Universal Robots PolyScope program: Short_LidToCamera.urp

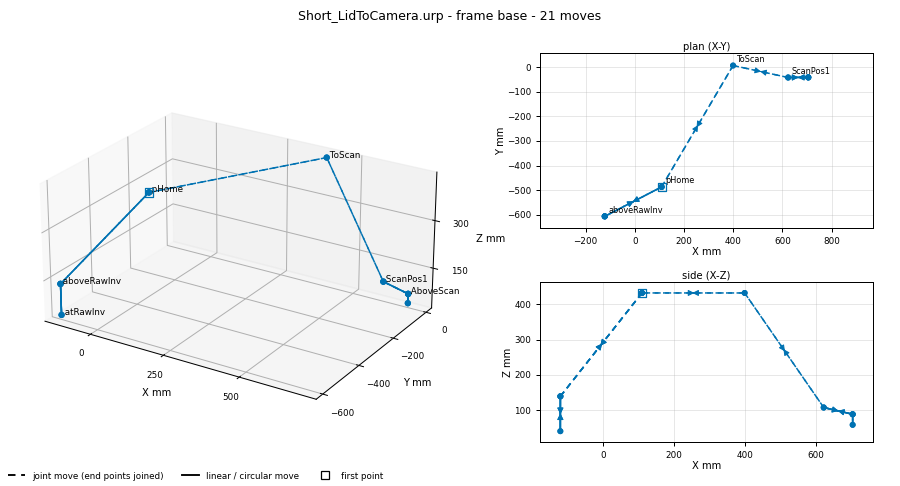
[picture p0: tool path of Short_LidToCamera.urp in frame base, 21 of 21 moves have a stored position in this frame; points joined in program order, loops and branches not executed]
Program Short_LidToCamera (installation=admin directory=/programs/THU_530PM/Final createdIn=3.8.0.61336 lastSavedIn=3.15.8.106339 robotSerialNumber=2015350926)
Calibrated DH parameters: a=[0, -0.425, -0.39225, 0, 0, 0]; d=[0.089159, 0, 0, 0.10915, 0.09465, 0.0823]; alpha=[1.570796, 0, 0, 1.570796, -1.570796, 0]; deltaTheta=[0, 0, 0, 0, 0, 0]
Robot Program (runOnlyOnce=true)
  Set DigitalOutput pin=digital_out[0]; digitalValue=0
  MoveJ speed 180 deg/s, acceleration 200 deg/s^2 (useActiveTCP=true)
    Waypoint pHome: TCP in base x=109.083 y=-486.882 z=431.849 mm, rx=0.0001 ry=3.1416 rz=-0.0001 rad; joints [89.992, -90.005, 90.008, -90.008, -90, -0.005] deg
    Call _adminLinearIndex1
    Waypoint aboveRawInv: TCP in base x=-121.786 y=-606.279 z=139.423 mm, rx=2.2213 ry=2.2177 rz=-0.001 rad; joints [68.458, -61.321, 99.13, -127.905, -89.867, 68.551] deg
  MoveL speed 250 mm/s, acceleration 1200 mm/s^2 (useActiveTCP=true) feature=Base
    Waypoint atRawInv: TCP in base x=-121.937 y=-606.364 z=40.769 mm, rx=2.2227 ry=2.216 rz=-0.0011 rad; joints [68.446, -51.912, 101.978, -140.169, -89.857, 68.619] deg
    Set DigitalOutput pin=digital_out[0]; digitalValue=1
    Wait Sleep waitTime=1
    Waypoint aboveRawInv: TCP in base x=-121.786 y=-606.279 z=139.423 mm, rx=2.2213 ry=2.2177 rz=-0.001 rad; joints [68.458, -61.321, 99.13, -127.905, -89.867, 68.551] deg
  MoveJ speed 180 deg/s, acceleration 200 deg/s^2 (useActiveTCP=true)
    Waypoint pHome: TCP in base x=109.083 y=-486.882 z=431.849 mm, rx=0.0001 ry=3.1416 rz=-0.0001 rad; joints [89.992, -90.005, 90.008, -90.008, -90, -0.005] deg
  Call _adminLinearIndex1
  MoveJ speed 60 deg/s, acceleration 80 deg/s^2 (useActiveTCP=true)
    Waypoint ToScan: TCP in base x=399.431 y=6.288 z=431.784 mm, rx=0 ry=-3.1415 rz=0 rad; joints [165.046, -103.944, 102.123, -88.173, -90.001, 75.046] deg
    Waypoint ScanPos1: TCP in base x=623.056 y=-42.326 z=107.794 mm, rx=0.0456 ry=-3.1308 rz=0.0038 rad; joints [166.086, -57.904, 99.074, -130.624, -90.289, 74.42] deg
  MoveL speed 250 mm/s, acceleration 1200 mm/s^2 (useActiveTCP=true) feature=Base
    Waypoint AboveScan: TCP in base x=704.91 y=-41.789 z=88.68 mm, rx=0.0458 ry=-3.1307 rz=0.0039 rad; joints [167.748, -47.56, 83.623, -125.504, -90.275, 76.074] deg
    Waypoint AtScan: TCP in base x=704.921 y=-41.77 z=58.801 mm, rx=0.0456 ry=-3.1306 rz=0.0038 rad; joints [167.749, -45.085, 84.321, -128.675, -90.272, 76.08] deg
    Set DigitalOutput pin=digital_out[0]; digitalValue=0
    Wait Sleep waitTime=1
    Waypoint AboveScan: TCP in base x=704.91 y=-41.789 z=88.68 mm, rx=0.0458 ry=-3.1307 rz=0.0039 rad; joints [167.748, -47.56, 83.623, -125.504, -90.275, 76.074] deg
    Waypoint ScanPos1: TCP in base x=623.056 y=-42.326 z=107.794 mm, rx=0.0456 ry=-3.1308 rz=0.0038 rad; joints [166.086, -57.904, 99.074, -130.624, -90.289, 74.42] deg
    Script file /programs/THU_530PM/vision_pc_modbus.script
      | pc_ip = "10.241.34.37"
      | pc_port = 30002
      | 
      | connection = socket_open(pc_ip, pc_port, "vision_socket")
      | 
      | if (connection):
      |     socket_send_string("run_vision", "vision_socket")
      |     socket_close("vision_socket")
      | end
      | 
      | timeout = 15.0
      | elapsed =0.0
      | visionResult = 0
      | while visionResult == 0 and elapsed < timeout:
      |          sync()
      |          sleep(0.2)
      |          elapsed = elapsed + 0.2
      |          visionResult = modbus_get_signal_status ("vision_result")
      |          sync()
      | end
    Wait Sleep waitTime=2
  MoveJ speed 60 deg/s, acceleration 80 deg/s^2 (useActiveTCP=true)
    Waypoint AboveScan: TCP in base x=704.91 y=-41.789 z=88.68 mm, rx=0.0458 ry=-3.1307 rz=0.0039 rad; joints [167.748, -47.56, 83.623, -125.504, -90.275, 76.074] deg
    Waypoint AtScan: TCP in base x=704.921 y=-41.77 z=58.801 mm, rx=0.0456 ry=-3.1306 rz=0.0038 rad; joints [167.749, -45.085, 84.321, -128.675, -90.272, 76.08] deg
    Set DigitalOutput pin=digital_out[0]; digitalValue=1
    Wait Sleep waitTime=1
    Waypoint AboveScan: TCP in base x=704.91 y=-41.789 z=88.68 mm, rx=0.0458 ry=-3.1307 rz=0.0039 rad; joints [167.748, -47.56, 83.623, -125.504, -90.275, 76.074] deg
  MoveJ speed 60 deg/s, acceleration 80 deg/s^2 (useActiveTCP=true)
    Waypoint ScanPos1: TCP in base x=623.056 y=-42.326 z=107.794 mm, rx=0.0456 ry=-3.1308 rz=0.0038 rad; joints [166.086, -57.904, 99.074, -130.624, -90.289, 74.42] deg
    Waypoint ToScan: TCP in base x=399.431 y=6.288 z=431.784 mm, rx=0 ry=-3.1415 rz=0 rad; joints [165.046, -103.944, 102.123, -88.173, -90.001, 75.046] deg
    Waypoint pHome: TCP in base x=109.083 y=-486.882 z=431.849 mm, rx=0.0001 ry=3.1416 rz=-0.0001 rad; joints [89.992, -90.005, 90.008, -90.008, -90, -0.005] deg
    Waypoint aboveRawInv: TCP in base x=-121.786 y=-606.279 z=139.423 mm, rx=2.2213 ry=2.2177 rz=-0.001 rad; joints [68.458, -61.321, 99.13, -127.905, -89.867, 68.551] deg
  MoveL speed 250 mm/s, acceleration 1200 mm/s^2 (useActiveTCP=true) feature=Base
    Waypoint atRawInv: TCP in base x=-121.937 y=-606.364 z=40.769 mm, rx=2.2227 ry=2.216 rz=-0.0011 rad; joints [68.446, -51.912, 101.978, -140.169, -89.857, 68.619] deg
    Set DigitalOutput pin=digital_out[0]; digitalValue=0
    Wait Sleep waitTime=1
    Waypoint aboveRawInv: TCP in base x=-121.786 y=-606.279 z=139.423 mm, rx=2.2213 ry=2.2177 rz=-0.001 rad; joints [68.458, -61.321, 99.13, -127.905, -89.867, 68.551] deg
  MoveJ speed 180 deg/s, acceleration 200 deg/s^2 (useActiveTCP=true)
    Waypoint pHome: TCP in base x=109.083 y=-486.882 z=431.849 mm, rx=0.0001 ry=3.1416 rz=-0.0001 rad; joints [89.992, -90.005, 90.008, -90.008, -90, -0.005] deg
SubProgram  [hidden by the author, left out]
SubProgram _adminLinearIndex1 [hidden by the author, left out]
